VAR_GLOBAL
	
	(* Selector*)
	stSelector	:	ST_Selector;
	stSelector2	:	ST_Selector;
	
	(* Cooler shaker *)
	stTECCtrl	: ARRAY[1..3] OF	ST_TECControl;
	stTECStatus	: ARRAY[1..3] OF	ST_TECStatus;
	
	stRegProp1	:	ST_Proportionair;
	stRegProp2	:	ST_Proportionair;
	stRegProp3	:	ST_Proportionair;
	stRegProp4	:	ST_Proportionair;
	
	(* Shakers *)
	stShaker01	:	ST_Shaker;
	stShaker02	:	ST_Shaker;
	stShaker03	:	ST_Shaker;
	stShaker04	:	ST_Shaker;
	
	(* Minitti Manifold *)
	stGasMani	:	ST_M3GasManifold;
	
	(* ALI *)
	stALI	:	ST_ALI;

END_VAR

(* stored: Version 1.1.0.1, ProductVersion 3.1.4020.12
   GVL GVL_Devices: Id {c147c728-648e-463f-984d-4f986cb4ad03} *)
